{attribute 'GeneratedUsingTerminal: EL6695-0002-0001'}
{attribute addProperty BoxType "EL6695-0002-0001"}
{attribute addProperty Id "EtcSlaveTerminalBaseSYNC_InputsAT %I*SYNC_Inputs_1DE69B903IO_InputsEMPTY_STRUCTURE0IO_OutputsEMPTY_STRUCTURE0WcStateAT %I*WcState_9091E0EB2InfoDataAT %I*InfoData_90184F0C16"}
{attribute addProperty CRC "2583790553"}
{attribute addProperty Size "21"}
TYPE EL6695_9A0183D9 EXTENDS EtcSlaveTerminalBase :
STRUCT
	{attribute addProperty Name "SYNC_Inputs"}
	SYNC_Inputs : SYNC_Inputs_1DE69B90;
	{attribute addProperty Name "IO_Inputs"}
	IO_Inputs : EMPTY_STRUCTURE;
	{attribute addProperty Name "IO_Outputs"}
	IO_Outputs : EMPTY_STRUCTURE;
	{attribute addProperty Name "WcState"}
	WcState : WcState_9091E0EB;
	{attribute addProperty Name "InfoData"}
	InfoData : InfoData_90184F0C;
END_STRUCT
END_TYPE

(* stored: Version 1.2.0.0, ProductVersion 3.1.4024.9
   DUT EL6695_9A0183D9: Id {a9f6be97-6a90-4e62-aa4b-8873b626a758} *)
